FUNCTION_BLOCK ASRT_SRT_TO_SR_AE (* Composite FB for convert ASRT to ASR + AE *)
  (* Standard: 61499-2; Description: Copyright (c) 2026 HR Agrartechnik GmbH This program and the accompanying materials are made available under the terms of the Eclipse Public License 2.0 which is available at https://www.eclipse.org/legal/epl-2.0/ SPDX-License-Identifier: EPL-2.0 *)
  (* Version 1.0, 2026-09-06, Franz Höpfinger, HR Agrartechnik GmbH *)
  PACKAGE adapter::conversion::unidirectional;
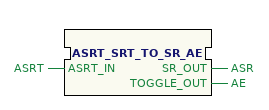
  SOCKETS
    ASRT_IN : adapter::types::unidirectional::ASRT; (* Adapter Input *)
  END_SOCKETS
  PLUGS
    SR_OUT : adapter::types::unidirectional::ASR; (* Set/Reset Output *)
    TOGGLE_OUT : adapter::types::unidirectional::AE; (* Toggle / Switch output *)
  END_PLUGS
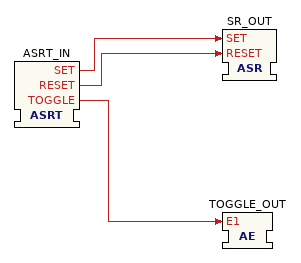
  EVENT_CONNECTIONS
    ASRT_IN.SET TO SR_OUT.SET;
    ASRT_IN.RESET TO SR_OUT.RESET;
    ASRT_IN.TOGGLE TO TOGGLE_OUT.E1;
  END_CONNECTIONS
END_FUNCTION_BLOCK
